PROGRAM MAIN
VAR
    (* 功能块 *)
    axis1: AXIS_REF;    (* 轴引用 *)

    (* 功能块 *)
    MCPower : MC_Power; (* 电机上电/下电控制功能块 *)
    MCJog   : MC_Jog;   (* 点动控制功能块 *)
	fbMoveCyclicPosition :MC_MoveRelative;
    fbMoveAbs      : MC_MoveAbsolute; // 定义绝对位置运动功能块
	MC_JOG :MC_JOG;


END_VAR

(* 使用速度控制 

*)

MCPower(Enable := TRUE,
		Enable_Positive := TRUE,
		Enable_Negative := TRUE,
		Override := 100,
		Axis  := axis1,
);
// 运动到绝对位置


//fbMoveCyclicPosition(Axis := axis1,Execute := TRUE, Distance:=3000,Velocity := 3000);

END_PROGRAM

(* stored: Version 1.1.0.1, ProductVersion 3.1.4024.12
   POU MAIN: Id {4404c240-9f3d-4bc8-84fa-e178cd1bb481}, SpecialFunc None *)
